(* IEC 61131-3 sources: repolevel_ST_code_completion/dataset/project_code/轴控/FB105_轴控制集/FB50_虚轴控制/FB101_功能块/F04_轴控操作, 6 files *)

(* ---- FB_读写ECT参数.st ---- *)
FUNCTION_BLOCK FB_读写ECT参数
VAR_INPUT
      Excute: BOOL;
      rWritePara1: REAL;
      rWritePara2: REAL;
      rWritePara3: REAL;

      SlaveAddr: UINT;

      SubIndexPara1: USINT;
      IndexPara1: UINT;
      SubIndexPara2: USINT;
      IndexPara2: UINT;
      SubIndexPara3: USINT;
      IndexPara3: UINT;

      SubIndexVel: USINT;
      IndexVel: UINT;
      SubIndexTou: USINT;
      IndexTou: UINT;
END_VAR
VAR_OUTPUT
      rReadPara1: REAL;
      rReadPara2: REAL;
      rReadPara3: REAL;
      rActVel:    REAL;
      rActTouque: REAL;
END_VAR
VAR
	BLINK0: BLINK;

	SMC3_ETC_ReadParameter_CoE_Para1: SMC3_ETC_ReadParameter_CoE;
	SMC3_ETC_ReadParameter_CoE_Para2: SMC3_ETC_ReadParameter_CoE;
	SMC3_ETC_ReadParameter_CoE_Para3: SMC3_ETC_ReadParameter_CoE;
	SMC3_ETC_ReadParameter_CoE_Vel:   SMC3_ETC_ReadParameter_CoE;
	SMC3_ETC_ReadParameter_CoE_Tou:   SMC3_ETC_ReadParameter_CoE;

	SMC3_ETC_WriteParameter_CoE_Para1: SMC3_ETC_WriteParameter_CoE;
	SMC3_ETC_WriteParameter_CoE_Para2: SMC3_ETC_WriteParameter_CoE;
	SMC3_ETC_WriteParameter_CoE_Para3: SMC3_ETC_WriteParameter_CoE;
	SMC3_ETC_WriteParameter_CoE_Vel:   SMC3_ETC_WriteParameter_CoE;
	SMC3_ETC_WriteParameter_CoE_Tou:   SMC3_ETC_WriteParameter_CoE;

    ReadPara1			      : DWORD;
	ReadPara2		          : DWORD;
	ReadPara3			      : DWORD;
	WritePara1			      : DWORD;
	WritePara2		          : DWORD;
	WritePara3			      : DWORD;

	ReadActVel			      : INT;
	ReadActTouque		      : INT;

END_VAR

VAR_IN_OUT
	AxisName: SM3_Drive_ETC.AXIS_REF_ETC_SM3;
END_VAR

BLINK0(ENABLE:= Excute, TIMELOW:= T#500MS, TIMEHIGH:= T#500MS, OUT=> );

IF rReadPara1<>rWritePara1 AND Excute THEN
	SMC3_ETC_WriteParameter_CoE_Para1.xExecute:=TRUE;
	ELSE
	SMC3_ETC_WriteParameter_CoE_Para1.xExecute:=FALSE;
END_IF
IF rReadPara2<>rWritePara2 AND Excute THEN
	SMC3_ETC_WriteParameter_CoE_Para2.xExecute:=TRUE;
	ELSE
	SMC3_ETC_WriteParameter_CoE_Para2.xExecute:=FALSE;
END_IF
IF rReadPara3<>rWritePara3 AND Excute THEN
	SMC3_ETC_WriteParameter_CoE_Para3.xExecute:=TRUE;
	ELSE
	SMC3_ETC_WriteParameter_CoE_Para3.xExecute:=FALSE;
END_IF

rReadPara1:=DWORD_TO_REAL(ReadPara1);
rReadPara2:=DWORD_TO_REAL(ReadPara2);
rReadPara3:=DWORD_TO_REAL(ReadPara3);
rActVel:=DWORD_TO_REAL(ReadActVel);
rActTouque:=DWORD_TO_REAL(ReadActTouque);

WritePara1:=REAL_TO_DWORD(rWritePara1);
WritePara2:=REAL_TO_DWORD(rWritePara2);
WritePara3:=REAL_TO_DWORD(rWritePara3);

(*读参数*)
SMC3_ETC_ReadParameter_CoE_Para1(
	xExecute:= BLINK0.OUT,
	xAbort:= ,
	uiIndex:= IndexPara1,
	usiSubIndex:= SubIndexPara1,
	Axis:= AxisName,
	xDone=> ,
	xBusy=> ,
	xError=> ,
	usiDataLength=> ,
	dwValue=> ADR(ReadPara1),
	dwErrorCode=> ,
	eError=> );

SMC3_ETC_ReadParameter_CoE_Para2(
	xExecute:= BLINK0.OUT,
	xAbort:= ,
	uiIndex:= IndexPara2,
	usiSubIndex:= SubIndexPara2,
	Axis:= AxisName,
	xDone=> ,
	xBusy=> ,
	xError=> ,
	usiDataLength=> ,
	dwValue=> ADR(ReadPara2),
	dwErrorCode=> ,
	eError=> );

SMC3_ETC_ReadParameter_CoE_Para3(
	xExecute:= BLINK0.OUT,
	xAbort:= ,
	uiIndex:= IndexPara3,
	usiSubIndex:= SubIndexPara3,
	Axis:= AxisName,
	xDone=> ,
	xBusy=> ,
	xError=> ,
	usiDataLength=> ,
	dwValue=> ADR(ReadPara3),
	dwErrorCode=> ,
	eError=> );

SMC3_ETC_ReadParameter_CoE_Vel(
	xExecute:= BLINK0.OUT,
	xAbort:= ,
	uiIndex:= IndexVel,
	usiSubIndex:= SubIndexVel,
	Axis:= AxisName,
	xDone=> ,
	xBusy=> ,
	xError=> ,
	usiDataLength=> ,
	dwValue=> ADR(ReadActVel),
	dwErrorCode=> ,
	eError=> );

SMC3_ETC_ReadParameter_CoE_Tou(
	xExecute:= BLINK0.OUT,
	xAbort:= ,
	uiIndex:= IndexTou,
	usiSubIndex:= SubIndexTou,
	Axis:= AxisName,
	xDone=> ,
	xBusy=> ,
	xError=> ,
	usiDataLength=> ,
	dwValue=> ADR(ReadActTouque),
	dwErrorCode=> ,
	eError=> );

(*写参数*)
SMC3_ETC_WriteParameter_CoE_Para1(
	xExecute:= ,
	xAbort:= ,
	uiIndex:= IndexPara1,
	usiSubIndex:= SubIndexPara1,
	usiDataLength:= DWORD_TO_USINT(SIZEOF(WritePara1)),
	dwValue:= ADR(WritePara1),
	Axis:= AxisName,
	xDone=> ,
	xBusy=> ,
	xError=> ,
	dwErrorCode=> ,
	eError=> );

SMC3_ETC_WriteParameter_CoE_Para2(
	xExecute:= ,
	xAbort:= ,
	uiIndex:= IndexPara2,
	usiSubIndex:= SubIndexPara2,
	usiDataLength:= DWORD_TO_USINT(SIZEOF(WritePara2)),
	dwValue:= ADR(WritePara2),
	Axis:= AxisName,
	xDone=> ,
	xBusy=> ,
	xError=> ,
	dwErrorCode=> ,
	eError=> );

SMC3_ETC_WriteParameter_CoE_Para3(
	xExecute:= ,
	xAbort:= ,
	uiIndex:= IndexPara3,
	usiSubIndex:= SubIndexPara3,
	usiDataLength:= DWORD_TO_USINT(SIZEOF(WritePara3)),
	dwValue:= ADR(WritePara3),
	Axis:= AxisName,
	xDone=> ,
	xBusy=> ,
	xError=> ,
	dwErrorCode=> ,
	eError=> );

(* ---- FB_轴停止触发块.st ---- *)
FUNCTION_BLOCK FB_轴停止触发块
VAR_IN_OUT
	StopExcute: BOOL;
END_VAR
VAR
	TON0: TON;
END_VAR

TON0(IN:= StopExcute, PT:= T#0.3S, Q=> , ET=> );

IF TON0.Q THEN
	StopExcute:=FALSE;
END_IF

(* ---- FB_轴回零.st ---- *)
FUNCTION_BLOCK FB_轴回零
VAR_INPUT
	Excute: BOOL;
	InputSigle: BOOL;
	Emergency: BOOL;
	OffersetDistance: LREAL;
	OffersetVel: LREAL;
	HomeVel: LREAL;
END_VAR

VAR_OUTPUT
	HomeBusy: BOOL;
	HomeDone: BOOL;
	HomeError: BOOL;
END_VAR
VAR
	R_TRIG0: R_TRIG;
	HoneStep: INT;
	MC_MoveRelative0: MC_MoveRelative;
	MC_Stop0: MC_Stop;
	MC_SetPosition0: MC_SetPosition;
	TON0: TON;
	TON1: TON;
	TON2: TON;
END_VAR

VAR_IN_OUT
	AxisName: SM3_BASIC.AXIS_REF_SM3;
END_VAR

MC_MoveRelative0(
	Axis:= AxisName,
	Execute:= ,
	Distance:= ,
	Velocity:= ,
	Acceleration:= 99999999,
	Deceleration:= 99999999,
	Jerk:= ,
	Done=> ,
	Busy=> ,
	CommandAborted=> ,
	Error=> ,
	ErrorID=> );

MC_Stop0(
	Axis:= AxisName,
	Execute:= ,
	Deceleration:= 1000000,
	Jerk:= ,
	Done=> ,
	Busy=> ,
	Error=> ,
	ErrorID=> );

MC_SetPosition0(
	Axis:= AxisName,
	Execute:= ,
	Position:= 0,
	Mode:= 0,
	Done=> ,
	Busy=> ,
	Error=> ,
	ErrorID=> );

IF HoneStep<>0 THEN
	HomeBusy:=TRUE;
	ELSE
	HomeBusy:=FALSE;
END_IF

IF MC_MoveRelative0.Error OR MC_Stop0.Error OR MC_SetPosition0.Error THEN
	HomeError:=TRUE;
	ELSE
	HomeError:=FALSE;
END_IF

IF Emergency THEN
	HoneStep:=0;
	MC_MoveRelative0.Execute:=FALSE;
	MC_Stop0.Execute:=FALSE;
	MC_SetPosition0.Execute:=FALSE;
	TON0(IN:= FALSE, );
	TON1(IN:= FALSE, );
	TON2(IN:= FALSE, );
	HomeBusy:=FALSE;
	HomeDone:=FALSE;
END_IF

R_TRIG0(CLK:= Excute, Q=> );

CASE HoneStep OF
	0:
	IF R_TRIG0.Q THEN
        HomeDone:=FALSE;
		HoneStep:=1;
	END_IF

	1:
	IF NOT InputSigle THEN
		MC_MoveRelative0.Velocity:=HomeVel;
		MC_MoveRelative0.Distance:=-9999999;
		MC_MoveRelative0.Execute:=TRUE;
		HoneStep:=5;
	END_IF
	IF InputSigle THEN
		MC_MoveRelative0.Velocity:=HomeVel;
		MC_MoveRelative0.Distance:=10;
		MC_MoveRelative0.Execute:=TRUE;
		HoneStep:=10;
	END_IF

	5:
	IF MC_MoveRelative0.Execute AND MC_MoveRelative0.Busy AND InputSigle THEN
		MC_MoveRelative0.Execute:=FALSE;
		HoneStep:=15;
	END_IF

	10:
	IF MC_MoveRelative0.Execute AND MC_MoveRelative0.Done THEN
		MC_MoveRelative0.Execute:=FALSE;
		HoneStep:=1;
	END_IF

	15:
	TON0(IN:= TRUE, PT:= T#0.1S, Q=> , ET=> );
	IF TON0.Q THEN
		MC_Stop0.Execute:=TRUE;
		IF MC_Stop0.Execute AND MC_Stop0.Done THEN
			MC_Stop0.Execute:=FALSE;
			TON0(IN:= FALSE, );
			HoneStep:=20;
		END_IF
	END_IF

	20:
	TON2(IN:= TRUE, PT:= T#0.1S, Q=> , ET=> );
	IF TON2.Q THEN
		MC_SetPosition0.Execute:=TRUE;
		IF MC_SetPosition0.Execute AND MC_SetPosition0.Done THEN
			MC_SetPosition0.Execute:=FALSE;
			TON2(IN:= FALSE, );
			HoneStep:=25;
		END_IF
	END_IF

	25:
	TON1(IN:= TRUE, PT:= T#0.1S, Q=> , ET=> );
	IF TON1.Q THEN
		MC_MoveRelative0.Velocity:=OffersetVel;
		MC_MoveRelative0.Distance:=OffersetDistance;
		MC_MoveRelative0.Execute:=TRUE;
		IF MC_MoveRelative0.Execute AND MC_MoveRelative0.Done THEN
			MC_MoveRelative0.Execute:=FALSE;
			TON1(IN:= FALSE, );
			HoneStep:=30;
		END_IF
	END_IF

	30:
	HomeDone:=TRUE;
	HoneStep:=0;

END_CASE

(* ---- FB_轴控块.st ---- *)
FUNCTION_BLOCK FB_轴控块
VAR_INPUT
	Enable: BOOL;

	JogFor: BOOL;
	JogBack: BOOL;
	JogVelocity :LREAL;

	StopExcute: BOOL;
	ResetExcute: BOOL;

	AbsExcute: BOOL;
	AbsPosition: LREAL;
	AbsVelocity: LREAL;
	AbsAcceleration: LREAL;
	AbsDeceleration: LREAL;

	RelExcute: BOOL;
	RelPosition: LREAL;
	RelVelocity: LREAL;
	RelAcceleration: LREAL;
	RelDeceleration: LREAL;

	VelExcute: BOOL;
	VelVelocity: LREAL;

    InchForward: BOOL;
	InchBackward: BOOL;
	InchDistance: LREAL;
	InchVelocity: LREAL;
	InchAcceleration: LREAL;
	InchDeceleration: LREAL;

	SetPosExcute: BOOL;

	ReStartSlaveEx: BOOL;
END_VAR
VAR_OUTPUT
	EnableStatus: BOOL;
	StopDone: BOOL;
	AbsDone: BOOL;
	RelDone: BOOL;
	VelBusy: BOOL;
	InchBusy: BOOL;
	JogBusy: BOOL;
	AbsBusy: BOOL;
	RelBusy: BOOL;
	AxisStandstill: BOOL;
	AxisError: BOOL;
	AxisAccing: BOOL;
	AxisDecing: BOOL;
	FBErrorOccured: BOOL;
	Homing: BOOL;
	Stopping: BOOL;
	ErrorID: SMC_ERROR;

	SetPosDone: BOOL;

	bOperational: BOOL;
	eComState: SM3_Basic.SMC_CommunicationState;
	wComState: WORD;

	ReStartSlaveDone: BOOL;
END_VAR
VAR
	MC_Power0: MC_Power;
	MC_Jog0: MC_Jog;
	MC_Stop0: MC_Stop;
	MC_Reset0: MC_Reset;
	MC_MoveAbsolute0: MC_MoveAbsolute;
	MC_MoveRelative0: MC_MoveRelative;
	MC_MoveVelocity0: MC_MoveVelocity;
	MC_ReadStatus0: MC_ReadStatus;
	SMC_Inch0: SMC_Inch;
	MC_SetPosition0: MC_SetPosition;
	SMC_CheckAxisCommunication0: SMC_CheckAxisCommunication;
	SMC3_ReinitDrive0: SMC3_ReinitDrive;
END_VAR

VAR_IN_OUT
	AxisName: SM3_BASIC.AXIS_REF_SM3;
END_VAR

MC_Power0(
	Axis:= AxisName,
	Enable:= TRUE,
	bRegulatorOn:= Enable,
	bDriveStart:= TRUE,
	Status=> EnableStatus,
	bRegulatorRealState=> ,
	bDriveStartRealState=> ,
	Busy=> ,
	Error=> ,
	ErrorID=> );

MC_Jog0(
	Axis:= AxisName,
	JogForward:= JogFor,
	JogBackward:= JogBack,
	Velocity:= JogVelocity,
	Acceleration:= JogVelocity*10000,
	Deceleration:= JogVelocity*10000,
	Jerk:= ,
	Busy=> JogBusy,
	CommandAborted=> ,
	Error=> ,
	ErrorId=> );

MC_Stop0(
	Axis:= AxisName,
	Execute:= StopExcute,
	Deceleration:= 100000000,
	Jerk:= ,
	Done=> StopDone,
	Busy=> ,
	Error=> ,
	ErrorID=> );

MC_Reset0(
	Axis:= AxisName,
	Execute:= ResetExcute,
	Done=> ,
	Busy=> ,
	Error=> ,
	ErrorID=> );

MC_SetPosition0(
	Axis:= AxisName,
	Execute:= SetPosExcute,
	Position:= 0,
	Mode:= 0,
	Done=> SetPosDone,
	Busy=> ,
	Error=> ,
	ErrorID=> );

MC_MoveAbsolute0(
	Axis:= AxisName,
	Execute:= AbsExcute,
	Position:= AbsPosition,
	Velocity:= AbsVelocity,
	Acceleration:= AbsAcceleration,
	Deceleration:= AbsDeceleration,
	Jerk:= ,
	Direction:= ,
	Done=> AbsDone,
	Busy=> AbsBusy,
	CommandAborted=> ,
	Error=> ,
	ErrorID=> );

MC_MoveRelative0(
	Axis:= AxisName,
	Execute:= RelExcute,
	Distance:= RelPosition,
	Velocity:= RelVelocity,
	Acceleration:= RelAcceleration,
	Deceleration:= RelDeceleration,
	Jerk:= ,
	Done=> RelDone,
	Busy=> RelBusy,
	CommandAborted=> ,
	Error=> ,
	ErrorID=> );

MC_MoveVelocity0(
	Axis:= AxisName,
	Execute:= VelExcute,
	Velocity:= VelVelocity,
	Acceleration:= VelVelocity*10000,
	Deceleration:= VelVelocity*10000,
	Jerk:= ,
	Direction:= ,
	InVelocity=> ,
	Busy=> VelBusy,
	CommandAborted=> ,
	Error=> ,
	ErrorID=> );

MC_ReadStatus0(
	Axis:= AxisName,
	Enable:= TRUE,
	Valid=> ,
	Busy=> ,
	Error=> ,
	ErrorID=> ErrorID,
	Disabled=> ,
	Errorstop=> AxisError,
	Stopping=> Stopping,
	StandStill=> AxisStandstill,
	DiscreteMotion=> ,
	ContinuousMotion=> ,
	SynchronizedMotion=> ,
	Homing=> Homing,
	ConstantVelocity=> ,
	Accelerating=> AxisAccing,
	Decelerating=> AxisDecing,
	FBErrorOccured=> FBErrorOccured);

SMC_Inch0(
	Axis:= AxisName,
	InchForward:= InchForward,
	InchBackward:= InchBackward,
	Distance:= InchDistance,
	Velocity:= InchVelocity,
	Acceleration:= InchAcceleration,
	Deceleration:= InchDeceleration,
	Jerk:= ,
	Busy=> InchBusy,
	CommandAborted=> ,
	Error=> ,
	ErrorId=> );

SMC_CheckAxisCommunication0(
	Axis:= AxisName,
	bEnable:= TRUE,
	bValid=> ,
	bError=> ,
	eErrorID=> ,
	bOperational=> bOperational,
	eComState=> eComState,
	wComState=> wComState);

SMC3_ReinitDrive0(
	Axis:= AxisName,
	bExecute:= ReStartSlaveEx,
	bVirtual:= ,
	bDone=> ReStartSlaveDone,
	bBusy=> ,
	bError=> ,
	nErrorID=> );

(* ---- FB_轴点动块.st ---- *)
FUNCTION_BLOCK FB_轴点动块
VAR_INPUT
	bForward		:BOOL;
	bBackward	    :BOOL;
	bFast			:BOOL;
	rAcceleration	:REAL:=1000;
	rDeceleration	:REAL:=1000;
	rSlowVelocity	:REAL:=2;
	rFastVelocity	:REAL:=3;
	tiWaitTime		:TIME:=t#0ms;
	rTipDistance	:REAL:=0;
END_VAR
VAR_OUTPUT
	bDone	:BOOL;
	bBusy	:BOOL;
	bCommandAborted	:BOOL;
	bError	:BOOL;
END_VAR
VAR
	diState: DINT;
	MC_MoveRelative_1: MC_MoveRelative;
	T_WaitTime: TON;
	MC_MoveVelocity_1: MC_MoveVelocity;
	MC_Stop_1: MC_Stop;
	bForwardInternal: BOOL;
	bBackwardInternal: BOOL;
	bFastInternal: BOOL;
END_VAR
VAR_IN_OUT
	Axis: SM3_BASIC.AXIS_REF_SM3;
END_VAR

(*
IF NOT V_emergy THEN
	diState	:=100;
END_IF
*)

CASE diState OF
	0:	(* Wait for Start *)
		bBusy		:=FALSE;
		bError		:=FALSE;
		bCommandAborted	:=FALSE;
		IF bForward XOR bBackward THEN
			bDone		:=FALSE;
			bBusy		:=TRUE;
			bError		:=FALSE;
			bForwardInternal	:=bForward;
			bBackwardInternal	:=bBackward;
			bFastInternal		:=bFast;
			diState	:=1;
		END_IF

	1:	(* Check parameters - If no Wait time or TippDistance -> immediate move velocity  *)
		IF TIME_TO_DINT(tiWaitTime) = 0 THEN
			diState	:=5;
		ELSIF rTipDistance = 0 THEN
			diState	:=5;
		ELSE
			diState	:=2;
		END_IF

	2:	(* Tipp Distance *)
		IF bForwardInternal AND NOT bBackwardInternal THEN
			MC_MoveRelative_1.Distance		:=rTipDistance;
		ELSIF bBackwardInternal AND NOT bForwardInternal THEN
			MC_MoveRelative_1.Distance		:=rTipDistance * -1;
		ELSE
			bError		:=TRUE;
			diState	:=100;
		END_IF
		IF bFastInternal THEN
			MC_MoveRelative_1.Velocity	:=rFastVelocity;
		ELSE
			MC_MoveRelative_1.Velocity	:=rSlowVelocity;
		END_IF
		MC_MoveRelative_1.Acceleration	:=rAcceleration;
		MC_MoveRelative_1.Deceleration	:=rDeceleration;
		MC_MoveRelative_1(Execute:=TRUE , Distance:= , Velocity:= , Acceleration:= , Deceleration:= , Axis:=Axis , Done=> , CommandAborted=> , Error=> , ErrorID=> );
		diState	:=3;

	3:
		T_WaitTime(IN:=TRUE , PT:=tiWaitTime , Q=> , ET=> );
		MC_MoveRelative_1(Execute:=TRUE , Distance:= , Velocity:= , Acceleration:= , Deceleration:= , Axis:=Axis , Done=> , CommandAborted=> , Error=> , ErrorID=> );
		IF MC_MoveRelative_1.Done THEN
			MC_MoveRelative_1(Execute:=FALSE , Distance:= , Velocity:= , Acceleration:= , Deceleration:= , Axis:=Axis , Done=> , CommandAborted=> , Error=> , ErrorID=> );
			diState	:=4;
		ELSIF MC_MoveRelative_1.Error OR (Axis.nAxisState = 1)  THEN
			T_WaitTime(IN:=FALSE , PT:=tiWaitTime , Q=> , ET=> );
			bError		:=TRUE;
			diState	:=100;
		ELSIF MC_MoveRelative_1.CommandAborted THEN
			T_WaitTime(IN:=FALSE , PT:=tiWaitTime , Q=> , ET=> );
			bCommandAborted	:=TRUE;
			diState	:=100;
		END_IF

	4:
		T_WaitTime(IN:=TRUE , PT:=tiWaitTime , Q=> , ET=> );
		IF NOT (bForward XOR bBackward) THEN
			bDone		:=TRUE;
			T_WaitTime(IN:=FALSE , PT:=tiWaitTime , Q=> , ET=> );
			diState	:=0;
		ELSIF T_WaitTime.Q THEN
			T_WaitTime(IN:=FALSE , PT:=tiWaitTime , Q=> , ET=> );
			diState	:=5;
		END_IF

	5:
		IF NOT (bForward XOR bBackward) THEN
			diState	:=0;
		ELSIF bForwardInternal AND NOT bBackwardInternal THEN
			MC_MoveVelocity_1.Direction	:=positive;
		ELSIF bBackwardInternal AND NOT bForwardInternal THEN
			MC_MoveVelocity_1.Direction	:=negative;
		END_IF
		IF bFast THEN
			MC_MoveVelocity_1.Velocity	:=rFastVelocity;
		ELSE
			MC_MoveVelocity_1.Velocity	:=rSlowVelocity;
		END_IF
		MC_MoveVelocity_1.Acceleration		:=rAcceleration;
		MC_MoveVelocity_1.Deceleration	:=rDeceleration;
		diState	:=6;

	6:
		MC_MoveVelocity_1(Execute:=TRUE , Velocity:= , Acceleration:= , Deceleration:= , Direction:= , Axis:=Axis , InVelocity=> , CommandAborted=> , Error=> , ErrorID=> );
		IF (bForward <> bForwardInternal) OR bBackward <> bBackwardInternal THEN
			MC_Stop_1(Execute:=TRUE ,Deceleration:=rDeceleration , Axis:=Axis, Done=> , Error=> , ErrorID=> );
			diState	:=7;
		ELSIF MC_MoveVelocity_1.CommandAborted THEN
			bCommandAborted		:=TRUE;
			diState	:=100;
		ELSIF MC_MoveVelocity_1.Error THEN
			bError		:=TRUE;
			diState	:=100;
		ELSE
			IF bFastInternal<>bFast THEN
				IF bFast THEN
					MC_MoveVelocity_1.Velocity	:=rFastVelocity;
				ELSE
					MC_MoveVelocity_1.Velocity	:=rSlowVelocity;
				END_IF
				MC_MoveVelocity_1(Execute:=FALSE , Velocity:= , Acceleration:= , Deceleration:= , Direction:= , Axis:=Axis , InVelocity=> , CommandAborted=> , Error=> , ErrorID=> );
				bFastInternal	:=bFast;
			END_IF
		END_IF
	7:
		MC_Stop_1(Execute:=TRUE ,Deceleration:=rDeceleration , Axis:=Axis, Done=> , Error=> , ErrorID=> );
		IF MC_Stop_1.Done THEN
			MC_Stop_1(Execute:=FALSE ,Deceleration:=rDeceleration , Axis:=Axis, Done=> , Error=> , ErrorID=> );
			MC_MoveVelocity_1(Execute:=FALSE , Velocity:= , Acceleration:= , Deceleration:= , Direction:= , Axis:=Axis , InVelocity=> , CommandAborted=> , Error=> , ErrorID=> );
			bDone		:=TRUE;
			diState	:=0;
		ELSIF MC_Stop_1.Error THEN
			MC_Stop_1(Execute:=FALSE ,Deceleration:=rDeceleration , Axis:=Axis, Done=> , Error=> , ErrorID=> );
			MC_MoveVelocity_1(Execute:=FALSE , Velocity:= , Acceleration:= , Deceleration:= , Direction:= , Axis:=Axis , InVelocity=> , CommandAborted=> , Error=> , ErrorID=> );
			bError		:=TRUE;
			diState	:=100;
		END_IF

	100:	(* Error *)
		bBusy	:=FALSE;
		MC_MoveRelative_1(Execute:=FALSE, Axis:=Axis);
		MC_MoveVelocity_1(Execute:=FALSE , Axis:=Axis);
		MC_Stop_1(Execute:=FALSE, Axis:=Axis);
		IF NOT bForward AND NOT bBackward THEN
			diState	:=0;
		END_IF
END_CASE

(* ---- FB_轴通讯状态块.st ---- *)
FUNCTION_BLOCK FB_轴通讯状态块
VAR_INPUT
	Axis_bCommunication: BOOL;
	Axis_wCommunicationState: WORD;
END_VAR
VAR_OUTPUT
	EtherCATBusOK: BOOL;
END_VAR
VAR
END_VAR

EtherCATBusOK := (Axis_wCommunicationState = 100) AND Axis_bCommunication;
